{attribute 'pack_mode' := '1'}
TYPE ClearAllFaults EXTENDS IncomingMessage :
STRUCT
END_STRUCT
END_TYPE

(* stored: Version 1.1.0.1, ProductVersion 3.1.4022.12
   DUT ClearAllFaults: Id {55405d70-b786-464d-87e8-d127bb263ec5} *)
